PROGRAM MAIN
VAR
	_tcoDigitalSensorTests : TcoDigitalSensorTests;
	_tcoDigitalActuatorTests : TcoDigitalActuatorTests;
END_VAR

_tcoDigitalSensorTests.ProbeRun();
_tcoDigitalActuatorTests.ProbeRun();

END_PROGRAM

(* stored: Version 1.1.0.1, ProductVersion 3.1.4024.6
   POU MAIN: Id {32b68bc5-5a7d-02c8-20e5-0d5146c25300}, SpecialFunc None *)
